// TIA Portal V17 export
// export: Created 2021-12-03T08:13:08.4691203Z, ExportSetting WithDefaults, DisplayName Totally Integrated Automation Portal, DisplayVersion V17, DisplayName TIA Portal Openness, DisplayVersion V17, DisplayName TIA Portal Version Control Interface, DisplayVersion V17, DisplayName STEP 7 Professional, DisplayVersion V17, DisplayName STEP 7 Safety, DisplayVersion V17, DisplayName WinCC Advanced, DisplayVersion V17
FUNCTION "FC_Faults" : Void   // FC40, FBD
VERSION : 0.1
// stored: AutoNumber false, IsIECCheckEnabled false, UDAEnableTagReadback false
BEGIN

NETWORK
TITLE = Ошибка питания 24V
      AN    "GDB_Inputs".I_BrPow1Flt;
      =     "GDB_Faults".CirBrk24VFb.I_BrPow1Flt;
      AN    "GDB_Inputs".I_BrPow2Flt;
      =     "GDB_Faults".CirBrk24VFb.I_BrPow2Flt;
      AN    "GDB_Inputs".I_SitopPow1Flt;
      =     "GDB_Faults".CirBrk24VFb.I_SitopPow1Flt;
      AN    "GDB_Inputs".I_SitopPow2Flt;
      =     "GDB_Faults".CirBrk24VFb.I_SitopPow2Flt;

NETWORK
TITLE = Ошибка питания 220V
      AN    "GDB_Inputs".I_BrLigSrvFlt;
      =     "GDB_Faults".CirBrk220VFb.I_BrLigSrvFlt;
      AN    "GDB_Inputs".I_BrAccConFlt;
      =     "GDB_Faults".CirBrk220VFb.I_BrAccConFlt;
      AN    "GDB_Inputs".I_BrXRayUnitFlt;
      =     "GDB_Faults".CirBrk220VFb.I_BrXRayUnitFlt;
      AN    "GDB_Inputs".I_BrPowPlcFlt;
      =     "GDB_Faults".CirBrk220VFb.I_BrPowPlcFlt;
      AN    "GDB_Inputs".I_BrMod1PFlt;
      =     "GDB_Faults".CirBrk220VFb.I_BrMod1PFlt;

NETWORK
TITLE = Ошибка питания 380V
      AN    "GDB_Inputs".I_BrModFlt;
      =     "GDB_Faults".CirBrk380VFb.I_BrModFlt;
      AN    "GDB_Inputs".I_BrChilFlt;
      =     "GDB_Faults".CirBrk380VFb.I_BrChilFlt;
      AN    "GDB_Inputs".I_BrFrqConvFlt;
      =     "GDB_Faults".CirBrk380VFb.I_BrFrqConvFlt;

NETWORK
TITLE = Ошибки пускателей
      A     "FGDB_ContCtrl".ModCont400_Err;
      =     "GDB_Faults".FeedBackControl.ModCont400_Err;
      A     "FGDB_ContCtrl".ModCont230_Err;
      =     "GDB_Faults".FeedBackControl.ModCont230_Err;
      A     "FGDB_ContCtrl".ChillCont_Err;
      =     "GDB_Faults".FeedBackControl.ChillCont_Err;
      A     "FGDB_ContCtrl".AccCont_Err;
      =     "GDB_Faults".FeedBackControl.AccCont_Err;
      A     "FGDB_ContCtrl".ConvCont_Err;
      =     "GDB_Faults".FeedBackControl.ConvCont_Err;

NETWORK
TITLE = Аварийные кнопки и периметр
      AN    "FGDB_EmStpButton".P1EmStp_Sv;
      =     "GDB_Faults".EmStBt.P1EmStp_Sv;
      AN    "FGDB_EmStpButton".P2EmStp_Sv;
      =     "GDB_Faults".EmStBt.P2EmStp_Sv;
      AN    "FGDB_EmStpButton".P3EmStp_Sv;
      =     "GDB_Faults".EmStBt.P3EmStp_Sv;
      AN    "FGDB_EmStpButton".AccEmStp_Sv;
      =     "GDB_Faults".EmStBt.AccEmStp_Sv;
      AN    "FGDB_EmStpButton".DosimEmStp_Sv;
      =     "GDB_Faults".EmStBt.DosimEmStp_Sv;
      A     "FGDB_Safety_Perimeter".SPBreak;
      =     "GDB_Faults".EmStBt.PerOpnIllegal;

REGION Network 6: Ошибка частотного преобразователя
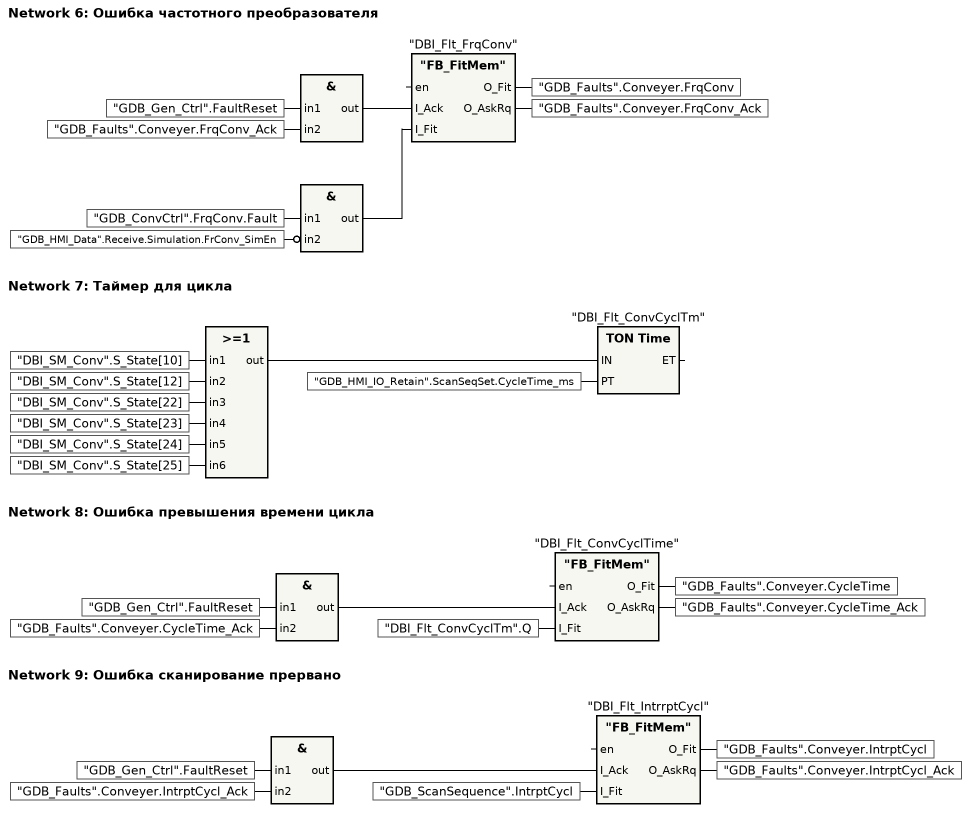
   "DBI_Flt_FrqConv"(I_Ack := "GDB_Gen_Ctrl".FaultReset AND "GDB_Faults".Conveyer.FrqConv_Ack,   // "FB_FitMem"
                     I_Fit := "GDB_ConvCtrl".FrqConv.Fault AND NOT "GDB_HMI_Data".Receive.Simulation.FrConv_SimEn,
                     O_Fit => "GDB_Faults".Conveyer.FrqConv,
                     O_AskRq => "GDB_Faults".Conveyer.FrqConv_Ack);
END_REGION

REGION Network 7: Таймер для цикла
   "DBI_Flt_ConvCyclTm".TON(IN := "DBI_SM_Conv".S_State[10] OR "DBI_SM_Conv".S_State[12] OR "DBI_SM_Conv".S_State[22] OR "DBI_SM_Conv".S_State[23] OR "DBI_SM_Conv".S_State[24] OR "DBI_SM_Conv".S_State[25],
                           PT := "GDB_HMI_IO_Retain".ScanSeqSet.CycleTime_ms);
END_REGION

REGION Network 8: Ошибка превышения времени цикла
   "DBI_Flt_ConvCyclTime"(I_Ack := "GDB_Gen_Ctrl".FaultReset AND "GDB_Faults".Conveyer.CycleTime_Ack,   // "FB_FitMem"
                          I_Fit := "DBI_Flt_ConvCyclTm".Q,
                          O_Fit => "GDB_Faults".Conveyer.CycleTime,
                          O_AskRq => "GDB_Faults".Conveyer.CycleTime_Ack);
END_REGION

REGION Network 9: Ошибка сканирование прервано
   "DBI_Flt_IntrrptCycl"(I_Ack := "GDB_Gen_Ctrl".FaultReset AND "GDB_Faults".Conveyer.IntrptCycl_Ack,   // "FB_FitMem"
                         I_Fit := "GDB_ScanSequence".IntrptCycl,
                         O_Fit => "GDB_Faults".Conveyer.IntrptCycl,
                         O_AskRq => "GDB_Faults".Conveyer.IntrptCycl_Ack);
END_REGION

NETWORK
TITLE = Ошибка сединения детекторной линейки
      AN    "GDB_DetLine".Status.ConOk;
      =     "GDB_Faults".DetLine.NotCon;


NETWORK
TITLE = Одна из ошибок
      O     "GDB_Faults".CirBrk24VFb.I_BrPow1Flt;
      O     "GDB_Faults".CirBrk24VFb.I_BrPow2Flt;
      O     "GDB_Faults".CirBrk24VFb.I_SitopPow1Flt;
      O     "GDB_Faults".CirBrk24VFb.I_SitopPow2Flt;
      O     "GDB_Faults".CirBrk220VFb.I_BrLigSrvFlt;
      O     "GDB_Faults".CirBrk220VFb.I_BrAccConFlt;
      O     "GDB_Faults".CirBrk220VFb.I_BrXRayUnitFlt;
      O     "GDB_Faults".CirBrk220VFb.I_BrPowPlcFlt;
      O     "GDB_Faults".CirBrk220VFb.I_BrMod1PFlt;
      O     "GDB_Faults".CirBrk380VFb.I_BrModFlt;
      O     "GDB_Faults".CirBrk380VFb.I_BrChilFlt;
      O     "GDB_Faults".CirBrk380VFb.I_BrFrqConvFlt;
      O     "GDB_Faults".FeedBackControl.ModCont400_Err;
      O     "GDB_Faults".FeedBackControl.ModCont230_Err;
      O     "GDB_Faults".FeedBackControl.ChillCont_Err;
      O     "GDB_Faults".FeedBackControl.AccCont_Err;
      O     "GDB_Faults".FeedBackControl.ConvCont_Err;
      O     "GDB_Faults".EmStBt.P1EmStp_Sv;
      O     "GDB_Faults".EmStBt.P2EmStp_Sv;
      O     "GDB_Faults".EmStBt.P3EmStp_Sv;
      O     "GDB_Faults".EmStBt.AccEmStp_Sv;
      O     "GDB_Faults".EmStBt.DosimEmStp_Sv;
      O     "GDB_Faults".EmStBt.PerOpnIllegal;
      O     "GDB_Faults".Conveyer.FrqConv;
      O     "GDB_Faults".Conveyer.CycleTime;
      O     "GDB_Faults".Conveyer.IntrptCycl;
      O     "GDB_Faults".DetLine.NotCon;
      =     "GDB_Faults".Com_Err;
END_FUNCTION
